(* Logix 5000 project; controller KTC_lab2 vendor 1 type 14 code 150 rev 30.11; software revision 30.00 *)

TASK MainTask (continuous, watchdog 500 ms) : MainProgram

MODULES
   Local : vendor 1 type 14 code 150 (Compact 0, rev 30.11)
      Counters : Embedded (Compact 3, rev 1.1, Output RPI 20 ms)
      Discrete_IO : Embedded (Compact 1, rev 3.1, Output RPI 20 ms)
      Analog_IO : Embedded (Compact 2, rev 1.1, Output RPI 80 ms)
END_MODULES

PROGRAM MainProgram   (* main routine MainRoutine *)
VAR
   PB0 : BOOL;   // NORMALY OPEN PUSH BUTTON 0
   PB1 : BOOL;   // NORMALLY CLOSED PUSH BUTTON 1
   PL1 : ALIAS FOR Local:1:O.Data.1;   // LIGHT 1
   PL3 : ALIAS FOR Local:1:O.Data.3;   // LIGHT 3
   PL4 : ALIAS FOR Local:1:O.Data.4;   // LIGHT 4
   PL5 : ALIAS FOR Local:1:O.Data.5;   // LIGHT 5
   PL6 : ALIAS FOR Local:1:O.Data.6;   // LIGHT 6
   PL7 : ALIAS FOR Local:1:O.Data.7;   // LIGHT 7
   SW4 : BOOL;   // SWITCH 4
   SW5 : BOOL;   // SWITCH 5 ALSO CONTROLS LIGHT 2 AND 4 SEE RUNG 4 AND 5
   SW6 : BOOL;   // SWITCH 6
   SW7 : BOOL;   // SWITCH 7
END_VAR

ROUTINE MainRoutine   (* ladder *)
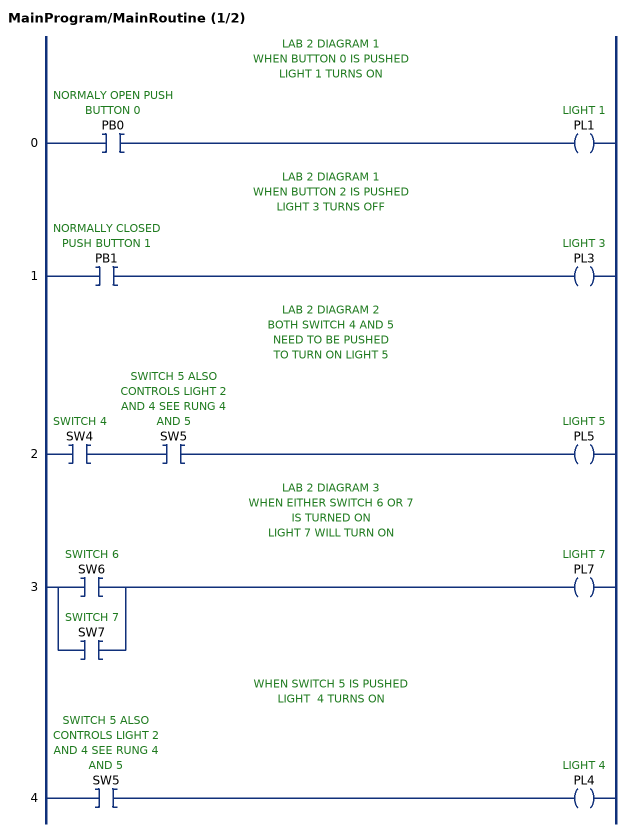
   // LAB 2 DIAGRAM 1
   // WHEN BUTTON 0 IS PUSHED
   // LIGHT 1 TURNS ON
   0: XIC(PB0)OTE(PL1);
   // LAB 2 DIAGRAM 1
   // WHEN BUTTON 2 IS PUSHED
   // LIGHT 3 TURNS OFF
   1: XIC(PB1)OTE(PL3);
   // LAB 2 DIAGRAM 2
   // BOTH SWITCH 4 AND 5
   // NEED TO BE PUSHED
   // TO TURN ON LIGHT 5
   2: XIC(SW4)XIC(SW5)OTE(PL5);
   // LAB 2 DIAGRAM 3
   // WHEN EITHER SWITCH 6 OR 7
   // IS TURNED ON
   // LIGHT 7 WILL TURN ON
   3: [XIC(SW6) ,XIC(SW7) ]OTE(PL7);
   // WHEN SWITCH 5 IS PUSHED
   // LIGHT  4 TURNS ON
   4: XIC(SW5)OTE(PL4);
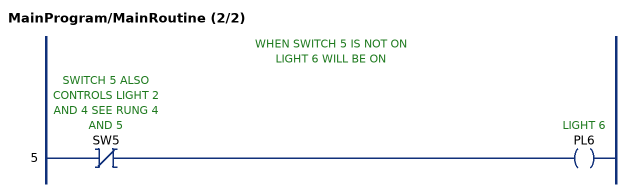
   // WHEN SWITCH 5 IS NOT ON
   // LIGHT 6 WILL BE ON
   5: XIO(SW5)OTE(PL6);
END_ROUTINE
END_PROGRAM
